{attribute addProperty BoxType "EL6090-0000-0016"}
{attribute addProperty Id "StatusAT %I*Status_F701F537162"}
{attribute addProperty CRC "599284590"}
{attribute addProperty SizeInBites "16"}
{attribute addProperty SizeInBytes "2"}
TYPE DIS_Inputs_23B85B6E :
STRUCT
	{attribute addProperty Name "Status"}
	Status AT %I* : Status_F701F537;
END_STRUCT
END_TYPE

(* stored: Version 1.2.0.0, ProductVersion 3.1.4024.9
   DUT DIS_Inputs_23B85B6E: Id {efec60ec-682e-4acd-93ba-6204981533b8} *)
